// SIMATIC STEP 7 (V5.x) project TEMA 13 EJERCICIO 27
// CPU: CPU313 C-2 DP(1)
// station: P_ADR_BUS
// station: Hardware
// station: Equipo SIMATIC 300
// program: Programa S7(1)

SYMBOL_TABLE
"FLANCOS"	DB 1	DB 1
"MANIOBRA"	DB 2	DB 2
"MARCHA"	I 0.0	BOOL
"PARO"	I 0.1	BOOL
"TERMICO"	I 0.2	BOOL
"Cycle Execution"	OB 1	OB 1
"M0T0R"	Q 0.0	BOOL
"LEDMARCHA"	Q 0.1	BOOL
"LEDDESCARGA"	Q 0.2	BOOL
"LEDPARO"	Q 0.3	BOOL
"LEDAVERIA"	Q 0.4	BOOL
END_SYMBOL_TABLE

DATA_BLOCK "FLANCOS"	// DB 1
VERSION : 0.1
  STRUCT
   M0 : BOOL ;
   M1 : BOOL ;
   M2 : BOOL ;
   M3 : BOOL ;
   M4 : BOOL ;
   M5 : BOOL ;
   M6 : BOOL ;
   M7 : BOOL ;
   M10 : BOOL ;
   M11 : BOOL ;
   M12 : BOOL ;
   M13 : BOOL ;
   M14 : BOOL ;
   M15 : BOOL ;
   M16 : BOOL ;
   M17 : BOOL ;
  END_STRUCT ;	
BEGIN
END_DATA_BLOCK

DATA_BLOCK "MANIOBRA"	// DB 2
VERSION : 0.1
  STRUCT
   MARCA0 : BOOL ;
   MARCA1 : BOOL ;
   MARCA3 : BOOL ;
   MARCA4 : BOOL ;
   MARCA5 : BOOL ;
   MARCA6 : BOOL ;
   MARCA7 : BOOL ;
  END_STRUCT ;	
BEGIN
END_DATA_BLOCK

ORGANIZATION_BLOCK "Cycle Execution"	// OB 1
TITLE = "Main Program Sweep (Cycle)"
//BOOMBEO DE GASOIL
VERSION : 0.1
VAR_TEMP
  OB1_EV_CLASS : BYTE ;	//Bits 0-3 = 1 (Coming event), Bits 4-7 = 1 (Event class 1)
  OB1_SCAN_1 : BYTE ;	//1 (Cold restart scan 1 of OB 1), 3 (Scan 2-n of OB 1)
  OB1_PRIORITY : BYTE ;	//Priority of OB Execution
  OB1_OB_NUMBR : BYTE ;	//1 (Organization block 1, OB1)
  OB1_RESERVED_1 : BYTE ;	//Reserved for system
  OB1_RESERVED_2 : BYTE ;	//Reserved for system
  OB1_PREV_CYCLE : INT ;	//Cycle time of previous OB1 scan (milliseconds)
  OB1_MIN_CYCLE : INT ;	//Minimum cycle time of OB1 (milliseconds)
  OB1_MAX_CYCLE : INT ;	//Maximum cycle time of OB1 (milliseconds)
  OB1_DATE_TIME : DATE_AND_TIME ;	//Date and time OB1 started
END_VAR
BEGIN
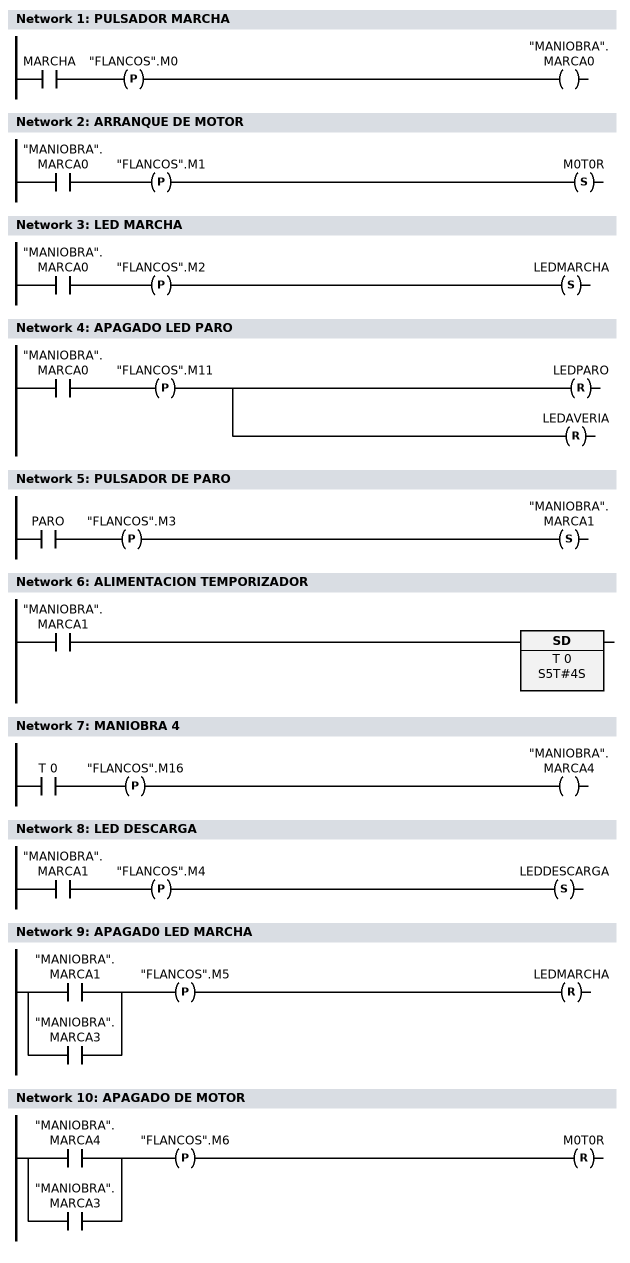
NETWORK
TITLE = PULSADOR MARCHA
      A     "MARCHA";
      FP    "FLANCOS".M0;
      =     "MANIOBRA".MARCA0;
NETWORK
TITLE = ARRANQUE DE MOTOR
      A     "MANIOBRA".MARCA0;
      FP    "FLANCOS".M1;
      S     "M0T0R";
NETWORK
TITLE = LED MARCHA
      A     "MANIOBRA".MARCA0;
      FP    "FLANCOS".M2;
      S     "LEDMARCHA";
NETWORK
TITLE = APAGADO LED PARO
      A     "MANIOBRA".MARCA0;
      FP    "FLANCOS".M11;
      R     "LEDPARO";
      R     "LEDAVERIA";
NETWORK
TITLE = PULSADOR DE PARO
//AL PULSAR EL MOTOR ENTRARA EN DESCARGA DURANTE 4 SEG.
      A     "PARO";
      FP    "FLANCOS".M3;
      S     "MANIOBRA".MARCA1;
NETWORK
TITLE = ALIMENTACION TEMPORIZADOR
      A     "MANIOBRA".MARCA1;
      L     S5T#4S;
      SD    T 0;
NETWORK
TITLE = MANIOBRA 4
      A     T 0;
      FP    "FLANCOS".M16;
      =     "MANIOBRA".MARCA4;
NETWORK
TITLE = LED DESCARGA
      A     "MANIOBRA".MARCA1;
      FP    "FLANCOS".M4;
      S     "LEDDESCARGA";
NETWORK
TITLE = APAGAD0 LED MARCHA
      A(;
      O     "MANIOBRA".MARCA1;
      O     "MANIOBRA".MARCA3;
      );
      FP    "FLANCOS".M5;
      R     "LEDMARCHA";
NETWORK
TITLE = APAGADO DE MOTOR
      A(;
      O     "MANIOBRA".MARCA4;
      O     "MANIOBRA".MARCA3;
      );
      FP    "FLANCOS".M6;
      R     "M0T0R";
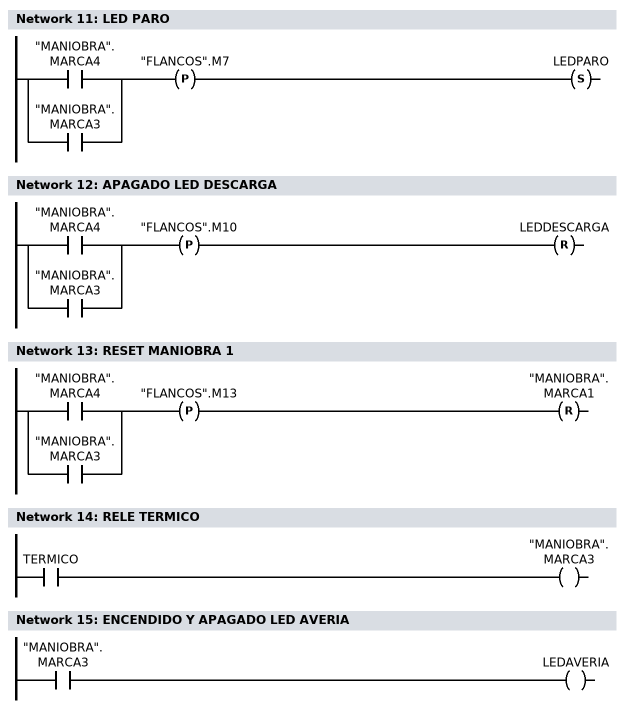
NETWORK
TITLE = LED PARO
      A(;
      O     "MANIOBRA".MARCA4;
      O     "MANIOBRA".MARCA3;
      );
      FP    "FLANCOS".M7;
      S     "LEDPARO";
NETWORK
TITLE = APAGADO LED DESCARGA
      A(;
      O     "MANIOBRA".MARCA4;
      O     "MANIOBRA".MARCA3;
      );
      FP    "FLANCOS".M10;
      R     "LEDDESCARGA";
NETWORK
TITLE = RESET MANIOBRA 1
      A(;
      O     "MANIOBRA".MARCA4;
      O     "MANIOBRA".MARCA3;
      );
      FP    "FLANCOS".M13;
      R     "MANIOBRA".MARCA1;
NETWORK
TITLE = RELE TERMICO 
//EN CASO DE AVERIA DESCONECTA TODO EL PROCESO;
//SE ENCIENDE LED AVERIA Y PARO.
//
      A     "TERMICO";
      =     "MANIOBRA".MARCA3;
NETWORK
TITLE = ENCENDIDO Y APAGADO LED AVERIA
//COMO ES UNA SIMULACION EL ELD PERMANECE EN ON CUANDO EL PULSADOR ESTE EN ON
      A     "MANIOBRA".MARCA3;
      =     "LEDAVERIA";
END_ORGANIZATION_BLOCK
